TYPE StrutturaGenericaQuotaAssi :
STRUCT
	X : LREAL := 20;
	Y : LREAL := 20;
	Z : LREAL := 20;
	J : LREAL := 2;

END_STRUCT
END_TYPE

(* stored: Version 1.1.0.1, ProductVersion 3.1.4024.11
   DUT StrutturaGenericaQuotaAssi: Id {1e443426-86e2-4440-bfeb-16ff6906e333} *)
